FUNCTION_BLOCK RingTokenConveyerCTL (* Composite Function Block Type *)
  (* Standard: 61499-2 *)
  (* Version 0.2, 2003-12-05, JHC, Rockwell Automation, Renamed from NEWCOMPFB. *)
  (* Version 0.1, 2002-01-08, JHC, Rockwell Automation, Added DLY FB as example. *)
  (* Version 0.0, 2000-05-27, JHC, Rockwell Automation *)
  (* Compiler header: package fb.rt.template; *)
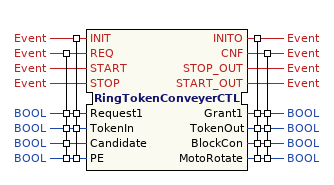
  EVENT_INPUT
    INIT WITH Request1, TokenIn, PE; (* Initialization Request *)
    REQ WITH Request1, TokenIn, Candidate, PE; (* Normal Execution Request *)
    START;
    STOP;
  END_EVENT
  EVENT_OUTPUT
    INITO WITH Grant1, TokenOut, MotoRotate, BlockCon; (* Initialization Confirm *)
    CNF WITH Grant1, TokenOut, BlockCon, MotoRotate; (* Execution Confirmation *)
    STOP_OUT;
    START_OUT;
  END_EVENT
  VAR_INPUT
    Request1 : BOOL; (* Input event qualifier *)
    TokenIn : BOOL;
    Candidate : BOOL;
    PE : BOOL;
  END_VAR
  VAR_OUTPUT
    Grant1 : BOOL; (* Output event qualifier *)
    TokenOut : BOOL;
    BlockCon : BOOL;
    MotoRotate : BOOL;
  END_VAR
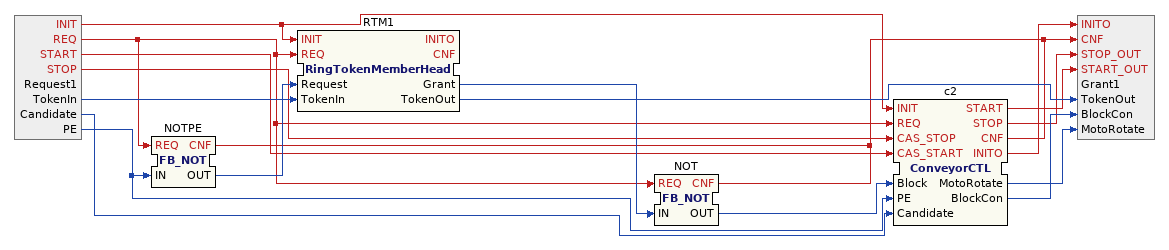
  FBS
    RTM1 : RingTokenMemberHead;
    c2 : ConveyorCTL;
    NOT : FB_NOT;
    NOTPE : FB_NOT;
  END_FBS
  EVENT_CONNECTIONS
    INIT TO RTM1.INIT;
    REQ TO RTM1.REQ;
    c2.START TO START_OUT;
    c2.STOP TO STOP_OUT;
    c2.CNF TO CNF;
    c2.INITO TO INITO;
    INIT TO c2.INIT;
    REQ TO c2.REQ;
    STOP TO c2.CAS_STOP;
    START TO c2.CAS_START;
    REQ TO NOTPE.REQ;
    NOTPE.CNF TO CNF;
    NOT.CNF TO CNF;
    REQ TO NOT.REQ;
  END_CONNECTIONS
  DATA_CONNECTIONS
    RTM1.Grant TO NOT.IN;
    NOT.OUT TO c2.Block;
    c2.MotoRotate TO MotoRotate;
    c2.BlockCon TO BlockCon;
    RTM1.TokenOut TO TokenOut;
    TokenIn TO RTM1.TokenIn;
    PE TO c2.PE;
    Candidate TO c2.Candidate;
    PE TO NOTPE.IN;
    NOTPE.OUT TO RTM1.Request;
  END_CONNECTIONS
END_FUNCTION_BLOCK
